(* IEC 61131-3 sources: PIDControlBackUpFolder/MyMPControl, 7 files *)

(* ---- Counter.st ---- *)
(* TODO: Add your comment here *)
FUNCTION_BLOCK Counter
	NumTimesIn := NumTimesIn + 1;
	IF NumTimesIn >= 1 THEN
		IF BoolExpIn = TRUE THEN
			BoolExpOut := FALSE;
		ELSE
			BoolExpOut := TRUE;
		END_IF
		NumTimesIn := 0;
	END_IF
	NumTimesOut := NumTimesIn;
END_FUNCTION_BLOCK

(* ---- DT_to_FIR.st ---- *)
FUNCTION_BLOCK DT_to_FIR

	FOR j := 0 TO SysOrder - 1 DO
		TempNum[j] := Num[j];
	END_FOR

	FOR j := 0 TO SysOrder DO
		TempDen[j] := Den[j];
	END_FOR

	FOR j:=0 TO SysOrder - 1 DO
		Num[j] := TempNum[SysOrder-j-1];
	END_FOR

	FOR j := 0 TO SysOrder DO
		Den[j] := TempDen [SysOrder-j];
	END_FOR

	FOR k := 0 TO TotalSamples - 1 DO

		IF k = 0 THEN
			StepResponse[k] := 0;

		ELSIF k = 1 THEN
			StepResponse[k] := Num[0] - (Den[1] * StepResponse[k - 1]);

		ELSIF k = 2 THEN
			StepResponse[k] := Num[0] + Num[1] - (Den[1] * StepResponse[k - 1] + Den[2] * StepResponse[k -2]);

		ELSIF k = 3 THEN
			StepResponse[k] := Num[0] + Num[1] + Num[2] - (Den[1] * StepResponse[k - 1] + Den[2] * StepResponse[k -2] + Den[3] * StepResponse[k - 3]);

		ELSIF k = 4 THEN
			StepResponse[k] := Num[0] + Num[1] + Num[2] + Num[3] - (Den[1] * StepResponse[k - 1] + Den[2] * StepResponse[k -2] + Den[3] * StepResponse[k - 3] + Den[4] * StepResponse[k - 4]);

		ELSE
			StepResponse[k] := Num[0] + Num[1] + Num[2] + Num[3] + Num[4] - (Den[1] * StepResponse[k - 1] + Den[2] * StepResponse[k -2] + Den[3] * StepResponse[k - 3] + Den[4] * StepResponse[k - 4] + Den[5] * StepResponse[k-5]);
		END_IF

	END_FOR

END_FUNCTION_BLOCK

(* ---- IDDone.st ---- *)
(* TODO: Add your comment here *)
FUNCTION_BLOCK IDDone
	IF DoneIn = TRUE OR DoneOnce > 0 THEN
		Done := TRUE;
		DoneOnce := 1;
	ELSE
		Done := FALSE;
	END_IF

END_FUNCTION_BLOCK

(* ---- LocalFunctions.fun ---- *)
FUNCTION_BLOCK DT_to_FIR

	VAR_INPUT
		SysOrder : INT;
		Num : ARRAY[0..4] OF REAL; (* Numerator coefficients b0..bM *)
		Den : ARRAY[0..5] OF REAL; (* Denominator coefficients a0..aN, with a0=1 *)
		TotalSamples : INT; (* Number of impulse response samples to generate, e.g. 400 *)
		StepHeight : REAL;
	END_VAR

	VAR_OUTPUT
		StepResponse : ARRAY[0..399] OF LREAL; (* Output FIR array (here fixed to 400 for MPC) *)
	END_VAR

	VAR
		k : INT;
		j : INT;
		TempNum : ARRAY[0..4] OF REAL;
		TempDen : ARRAY[0..5] OF REAL;
		den0 : REAL := 1;
		TempStep : LREAL;
	END_VAR

END_FUNCTION_BLOCK

FUNCTION_BLOCK SetTargetValue

	VAR_INPUT
		TargetValue : REAL;
		CurrentVelocity : REAL;
		newSetValue : BOOL;

	END_VAR

	VAR_OUTPUT
		TargetValueArray : ARRAY[0..199] OF LREAL;
	END_VAR

	VAR
		i : INT;
		InitVelocity : REAL;
	END_VAR

END_FUNCTION_BLOCK

FUNCTION_BLOCK Counter

	VAR_INPUT
		BoolExpIn : BOOL;
		NumTimesIn : REAL;
		newParam : {REDUND_UNREPLICABLE} BOOL;
	END_VAR

	VAR_OUTPUT
		BoolExpOut : BOOL;
		NumTimesOut : REAL;
	END_VAR

END_FUNCTION_BLOCK

FUNCTION_BLOCK IDDone

	VAR_OUTPUT
		Done :  BOOL;
	END_VAR

	VAR_INPUT
		DoneIn : BOOL; (**)
	END_VAR

	VAR_IN_OUT
		DoneOnce : INT;
	END_VAR

END_FUNCTION_BLOCK

(* ---- SetTargetValue.st ---- *)
FUNCTION_BLOCK SetTargetValue

	InitVelocity := CurrentVelocity;

	IF newSetValue = TRUE THEN

		FOR i := 0 TO 199 DO
			TargetValueArray[i] := ((TargetValue - InitVelocity) * i)/200.0 + InitVelocity;
		END_FOR

		newSetValue := FALSE;
	END_IF

END_FUNCTION_BLOCK

(* ---- Init.st ---- *)
PROGRAM _INIT

	MPControlParameters.MemMode := TRUE;
	MPControlParameters.CycleFactor := 1;
	MPControlParameters.NrDist := 0;
	MPControlParameters.PredictionHorizon := 50;
	MPControlParameters.ControlHorizon := 20;
	MPControlParameters.OutSamplesMerge := 1;
	MPControlParameters.OutOperatingPoint := 0.1;
	MPControlParameters.ActOperatingPoint := 0.0;
	MPControlParameters.WeightErrorExp := 0.0;
	MPControlParameters.WeightError := 1.0;
	MPControlParameters.OutMoveSuppression := 0.1;
	MPControlParameters.ActDeltaWeight := 0.2;
	MPControlParameters.FIRModel := FALSE;
	MPControlParameters.SoftConstraint := FALSE;
	MPControlParameters.OutDeltaMax := 1.0;
	MPControlParameters.OutDeltaMin := 0.0;
	MPControlParameters.OutMin := -0.5;
	MPControlParameters.OutMax := 0.5;
	MPControlParameters.PostCtrlDisable := FALSE;

	AxisParameters.Position := 10000000;
	AxisParameters.Velocity := 1000;
	AxisParameters.Acceleration := 1000;
	AxisParameters.Deceleration := 1000;
	AxisParameters.Jerk := 10000;

END_PROGRAM

(* ---- Variables.var ---- *)
VAR
	AxisBasic : MpAxisBasic;
	AxisParameters : MpAxisBasicParType;
	AxisBasicEnable : BOOL := TRUE;
	AxisBasicUpdate : BOOL;
	AxisBasicSimulate : BOOL;
	AxisBasicPower : BOOL;
	AxisBasicErrorReset : BOOL;
	AxisBasicHome : BOOL;
	AxisBasicMoveVelocity : BOOL;
	AxisBasicMoveAbsolute : BOOL;
	AxisBasicMoveAdditive : BOOL;
	AxisBasicStop : BOOL;
	AxisBasicJogPositive : BOOL;
	AxisBasicJogNegative : BOOL;
	AxisBasicLimitLoad : BOOL;
	AxisBasicReleaseBrake : BOOL;
	AxisBasicAutoTune : BOOL;
	CurrentTorque : REAL;
	CurrentPosition : LREAL;
	CurrentVelocity : REAL;
	SampleTime : REAL;
	SysRef : UDINT;
	TrueBlockTorque : BOOL := FALSE;
	TrueBlockAxis : BOOL := FALSE;
	TrueBlockMPC : BOOL := TRUE;
	TrueBlockMTIdent : BOOL := FALSE;
	i : USINT := 0;
	TorqueControl : MC_BR_TorqueControl;
	TorqueControlEnable : BOOL;
	TorqueControlInitData : BOOL;
	TorqueControlTorque : REAL;
	TorqueControlTorqueRamp : REAL := 0;
	TorqueControlPosMaxVelocity : REAL := 1000;
	TorqueControlNegMaxVelocity : REAL := -1000;
	TorqueControlAcceleration : REAL := 1000;
	TorqueControlJerk : REAL;
	TorqueControlAdvancedParameters : McAdvBrTorqueControlParType;
	TorqueControlStart : BOOL;
	TorqueControlStop : BOOL;
	OverrideControl : BOOL;
	MTIdent : MTIdentLSQ;
	MTIdentEnable : BOOL;
	MTIdentSystemOrder : USINT := 2; (*Note: Changing the system order also means that you have to change the array size of the function that converts the DTF to FIR for Num and Den*)
	MTIdentStepHeight : REAL := 0.05;
	MTIdentUpdate : BOOL;
	MTIdentPlantOutput : REAL;
	MTIdentStartIdentification : BOOL;
	MTIdentWeighingFactor : REAL := 0.95;
	MTIdentSetIDDone : BOOL;
	ReadActualPosition : MC_ReadActualPosition;
	ReadActualPositionEnable : BOOL := TRUE;
	ReadActualVelocity : MC_ReadActualVelocity;
	ReadActualVelocityEnable : BOOL := TRUE;
	PositionLow : MTFilterLowPass;
	PositionLowEnable : BOOL := TRUE;
	PositionLowType : MTFilterTypeEnum := 0;
	PositionLowOrder : USINT := 2;
	PositionLowCutFreq : REAL := 0.05;
	PositionLowUpdate : BOOL := TRUE;
	PositionLowIn : REAL;
	VelocityBandPass : MTFilterBandPass;
	VelocityBandPassEnable : BOOL := TRUE;
	VelocityBandPassType : MTFilterTypeEnum := 0;
	VelocityBandPassOrder : USINT := 2;
	VelocityBandPassCentreFreq : REAL := 100;
	VelocityBandPassBandwidth : REAL := 199.95;
	VelocityBandPassUpdate : BOOL := TRUE;
	VelocityBandPassIn : REAL;
	WaitTime : TIME := T#100ms;
	WaitSimulate : TON;
	WaitPower : TON;
	WaitLoopShape : TON;
	WaitMTIdentEnable : TON;
	WaitTorqueEnable : TON;
	WaitTorqueStart : TON;
	WaitMTIdentStart : TON;
	AlwaysTrue : BOOL := TRUE;
	ModelConversion : DT_to_FIR;
	ModelConversionTotalSamples : INT := 400;
	MPControl : MTMpcSisoLite;
	MPControlEnable : BOOL; (*Parameters*)
	MPControlParameters : MTMpcSisoParameterType;
	MPControlUpdate : BOOL;
	MPControlSetValue : DINT;
	MPControlActValue : LREAL;
	MPControlOutReference : LREAL;
	MPControlSetDr : DINT;
	MPControlActDr : LREAL;
	MPControlDisturbEnable : BOOL;
	MPControlSetValueArray : ARRAY[0..199] OF LREAL;
	MPControlTargetValueSetter : SetTargetValue;
	MPControlTargetValue : REAL;
	MPCBoolExp : BOOL;
	MPControlNumTimes : REAL;
	MPControlCounter : Counter;
	MPControlNewSetValue : BOOL;
	MPControlTorqueArraySize : INT := 4;
	MPControlTorqueValueArray : ARRAY[0..199] OF LREAL;
	MPControlPosition : INT := 200;
	NeedToRunMPC : BOOL := TRUE;
	MPControlPrevTargetValue : REAL;
	MPControlPrevVelocity : REAL;
	ReturnHome : MC_MoveAbsolute;
	ReturnHomeExecute : BOOL;
	ReturnHomePosition : LREAL := 0;
	ReturnHomeVelocity : REAL := 1;
	ReturnHomeAcceleration : REAL := 0.1;
	ReturnHomeDeceleration : REAL := 0.11;
	ReturnHomeJerk : REAL := 0.01;
	ReturnHomeDirection : McDirectionEnum := 10;
	ReturnHomeBufferMode : McBufferModeEnum;
	DoneOnce : INT;
	CheckDone : IDDone;
END_VAR
